(* IEC 61131-3 sources: generating_plc_code_with_llms/Code#1/Bard/first run, 20 files *)

(* ---- 14.st ---- *)
// 13.26s
// 2
FUNCTION FC1001(measuredValue: REAL, switchingValue: REAL, hysteresis: REAL): BOOL
VAR
previousOutput: BOOL; (* Flag indicating the previous output state )
switchingThreshold: REAL; ( Hysteresis-adjusted switching value *)

BEGIN
previousOutput := FALSE; (* Initialize previous output state to FALSE )
switchingThreshold := switchingValue * (1.0 - hysteresis / 100.0); ( Calculate the hysteresis-adjusted switching threshold *)

IF measuredValue >= switchingThreshold THEN
IF NOT previousOutput THEN
previousOutput := TRUE;
RETURN TRUE; (* Switch output on *)
END_IF;

RETURN previousOutput; (* Maintain output state *)
ELSE
IF previousOutput THEN
previousOutput := FALSE;
RETURN FALSE; (* Switch output off *)
END_IF;

RETURN previousOutput; (* Maintain output state *)
END_IF;
END_FUNCTION

(* ---- 15.st ---- *)
// 16.13s
// 1
FUNCTION FC1002(sensorInput: BOOL, manualSwitch: BOOL, hornOutput: BOOL, alarmOutput: BOOL, indicatorOutput: BOOL):
VAR
sensorState: BOOL; (* Flag indicating the current sensor state )
presenceTimer: TOF; ( Timer for object presence detection )
alarmEnabled: BOOL; ( Flag indicating whether the alarm is enabled *)

BEGIN
sensorState := sensorInput; (* Update sensor state *)

(* Update presence timer )
presenceTimer.IN := sensorState; ( Start/stop timer based on sensor state *)

(* Determine alarm state )
IF presenceTimer.Q AND presenceTimer.ET >= 3000 THEN
alarmEnabled := TRUE; ( Alarm condition met after 3 seconds )
ELSE
alarmEnabled := FALSE; ( Alarm condition not met or reset *)
END_IF;

(* Control outputs )
hornOutput := sensorState AND NOT alarmEnabled; ( Horn on for approach, off for alarm )
alarmOutput := alarmEnabled AND manualSwitch; ( Alarm on for alarm condition and manual switch on )
indicatorOutput := manualSwitch; ( Indicator on when manual switch is on *)
END_FUNCTION

VAR
  sensorInput: BOOL; (* Analog input value from ultrasonic sensor *)
  manualSwitch: BOOL; (* Input value from manual switch E_A *)
  hornOutput: BOOL; (* Output signal for horn P_HU *)
  alarmOutput: BOOL; (* Output signal for alarm P_AL *)
  indicatorOutput: BOOL; (* Output signal for indicator P1 *)

sensorInput := ReadAnalogInput(sensorInput);
manualSwitch := ReadInput(manualSwitchInput);

(* Call FC1002 to update outputs based on sensor input and manual switch *)
FC1002(sensorInput, manualSwitch, hornOutput, alarmOutput, indicatorOutput);

(* Control output devices based on updated output variables *)
WriteOutput(hornOutput, hornOutputDevice);
WriteOutput(alarmOutput, alarmOutputDevice);
WriteOutput(indicatorOutput, indicatorOutputDevice);

(* ---- 18.st ---- *)
// 7.53s
// 2
FUNCTION FC1003(inputValue: REAL; IN_MIN: REAL; IN_MAX: REAL; OUT_MIN: REAL; OUT_MAX: REAL): REAL
VAR
  rangeRatio: REAL; (* Ratio between input and output ranges *)
  scaledValue: REAL; (* Scaled input value *)

BEGIN
  (* Calculate range ratio *)
  rangeRatio := (OUT_MAX - OUT_MIN) / (IN_MAX - IN_MIN);

  (* Scale input value to output range *)
  scaledValue := (inputValue - IN_MIN) * rangeRatio;

  (* Adjust scaled value to output range limits *)
  IF scaledValue < OUT_MIN THEN
    scaledValue := OUT_MIN;
  ELSIF scaledValue > OUT_MAX THEN
    scaledValue := OUT_MAX;
  END_IF;

  (* Return scaled input value *)
  RETURN scaledValue;
END_FUNCTION

(* ---- 19.st ---- *)
// 9.82s
// 2
FUNCTION_BLOCK FB1005(
START: BOOL;
THICKNESS MD_1: BYTE;
V_MAX: REAL;
V_MIN: REAL;
D_MAX: BYTE;
D_MIN: BYTE;
)
VAR
currentThickness: REAL; (* Current thickness measurement )
largestThickness: REAL; ( Largest thickness measurement in current cycle )
smallestThickness: REAL; ( Smallest thickness measurement in current cycle )
rejectLight: BOOL; ( Flag indicating whether reject light is on *)

BEGIN
(* Initialize variables *)
largestThickness := 0.0;
smallestThickness := 0.0;
rejectLight := FALSE;

(* Continuously check for measurement start )
WHILE TRUE DO
IF START THEN
currentThickness := REAL(MD_1); ( Convert thickness value from flag double word *)

  (* Check for new largest or smallest thickness record *)
  IF currentThickness > largestThickness THEN
    largestThickness := currentThickness;
    D_MAX := MD_1; (* Update largest thickness output *)
  ELSIF currentThickness < smallestThickness THEN
    smallestThickness := currentThickness;
    D_MIN := MD_1;
  END_IF;

  (* Check for out-of-tolerance thickness *)
  IF currentThickness < V_MIN OR currentThickness > V_MAX THEN
    rejectLight := TRUE;

    (* Disable further measurement until restart *)
    START := FALSE;
  ELSE
    rejectLight := FALSE;
  END_IF;
END_IF;

(* Delay for 1 millisecond to avoid excessive processing *)
DELAY 0.001;
END_WHILE;
END_FUNCTION_BLOCK

VAR
  sensorS1: BOOL; (* Input signal from sensor S1 *)
  thicknessMD1: BYTE; (* Flag double word representing thickness measurement *)
  vMax: REAL; (* Maximum thickness tolerance *)
  vMin: REAL; (* Minimum thickness tolerance *)
  thicknessDMax: BYTE; (* Output flag double word for largest thickness *)
  thicknessDMin: BYTE; (* Output flag double word for smallest thickness *)

(* Call FB1005 to check plate thickness and update output variables *)
FB1005(sensorS1, thicknessMD1, vMax, vMin, thicknessDMax, thicknessDMin);

(* Update output devices based on output variables *)
WriteOutput(thicknessDMax, thicknessDMaxOutput);
WriteOutput(thicknessDMin, thicknessDMinOutput);

(* ---- 21.st ---- *)
// 14.54s
// 2
FUNCTION_BLOCK FB_BURNER(
  IN: BOOL;
  OVER_TEMP: BOOL;
  OIL_TEMP: BOOL;
  STAGE2: BOOL;
  RST: BOOL;
  PRE_HEAT_TIME: TIME;
  SAFETY_TIME: TIME;
  STAGE2_DELAY: TIME;
  MULTIPLE_IGNITION: BOOL;
  LOCKOUT_TIME: TIME;
  // Add other required parameters:
  PPR_IGNITION_TIME: TIME;
  PRE_VENTILATION_TIME: TIME;
  POST_IGNITION_TIME: TIME;
)
VAR
  // Internal states
  currentState: INT;
  lockOutTimer: TON;
  stage1Timer: TON;
  stage2Timer: TON;
  ignitionActive: BOOL;
  flameDetected: BOOL;
  error: INT;

BEGIN
  // Initialize variables
  lockOutTimer.IN := FALSE;
  stage1Timer.IN := FALSE;
  stage2Timer.IN := FALSE;
  ignitionActive := FALSE;
  flameDetected := FALSE;
  error := 0;

  // State machine transitions
  CASE currentState OF
    // Standby
    0: IF IN AND NOT OVER_TEMP THEN
        currentState := 1;
        PRE_HEAT := TRUE; // Start fuel oil warming
      END_IF;
    // Fuel oil warming
    1: IF OIL_TEMP THEN
        currentState := 2;
        ENGINE_ON := TRUE; // Start engine
        stage1Timer.IN := TRUE; // Start stage 1 timer
      ELSIF TIME_GT(TIME_DIFF(T_NOW(), START_TIME), PRE_HEAT_TIME) THEN
        error := 1;
        currentState := 10; // Go to error state
        FAIL := TRUE;
      END_IF;
    // Pre-ventilation
    2: IF TIME_GT(TIME_DIFF(T_NOW(), START_TIME), PRE_VENTILATION_TIME) THEN
        currentState := 3;
        IGNITION := TRUE; // Activate ignition
        ignitionActive := TRUE;
      ELSIF flameDetected THEN
        error := 3;
        currentState := 10; // Go to error state
        FAIL := TRUE;
      END_IF;
    // Ignition phase
    3: IF TIME_GT(TIME_DIFF(T_NOW(), START_TIME), PPR_IGNITION_TIME + SAFETY_TIME) THEN
        error := 4;
        currentState := 10; // Go to error state
        FAIL := TRUE;
      ELSIF flameDetected THEN
        currentState := 4;
        OIL_VALVE := TRUE; // Open oil valve
        ignitionActive := FALSE;
      END_IF;
    // Burning stage 1
    4: IF flameDetected THEN
        IF MULTIPLE_IGNITION AND NOT flameDetected THEN
          currentState := 3; // Restart ignition if flame breaks
        END_IF;
        IF STAGE2 AND TIME_GT(TIME_DIFF(T_NOW(), START_TIME), stage1Timer.PT + STAGE2_DELAY) THEN
          currentState := 5;
          stage2Timer.IN := TRUE; // Start stage 2 timer
        END_IF;
      ELSE
        error := 5;
        currentState := 10; // Go to error state
        FAIL := TRUE;
      END_IF;
    // Burning stage 2
    5: IF flameDetected THEN
        IF MULTIPLE_IGNITION AND NOT flameDetected THEN
          currentState := 3; // Restart ignition if flame breaks
        END_IF;
      ELSE
        error := 5;
        currentState := 10; // Go to error state
        FAIL := TRUE;
      END_IF;
    // Error state
    10: IF RST AND NOT OVER_TEMP THEN
        IF TIME_GT(TIME_DIFF(T_NOW(), START_TIME), LOCKOUT_TIME) THEN
          currentState := 0; // Reset and go to standby
        END_IF;
      ELSE
        lockOutTimer.IN := TRUE; // Start lockout timer
      END_IF;
  END_CASE;

  // Update outputs based on current state
  CASE currentState OF
    0: STATUS := 110;
    1: STATUS := 111;
    2: STATUS := 111;
    3: STATUS := 111;
    4: STATUS := 112;
    5: STATUS := 1

(* ---- 1.st ---- *)
//5.93s
//3
(* Program to manage two alarms *)

VAR
  xAlarm1: BOOL; (* Alarm 1 status *)
  xAlarm2: BOOL; (* Alarm 2 status *)
  xAllOn: BOOL; (* Set all alarms on *)
  xAllOff: BOOL; (* Set all alarms off *)

(* Main program *)
PROGRAM Main
BEGIN
  IF xAllOn THEN
    xAlarm1 := TRUE;
    xAlarm2 := TRUE;
  ELSIF xAllOff THEN
    xAlarm1 := FALSE;
    xAlarm2 := FALSE;
  END_IF;
END_PROGRAM

(* ---- 10.st ---- *)
//8.
// 2
(* Program to implement the sigmoid function *)

FUNCTION Sigmoid(x: REAL): REAL
BEGIN
  RETURN(1.0 / (1.0 + EXP(-x)));
END_FUNCTION

(* Main program *)
PROGRAM Main
VAR
  x: REAL; (* Input value *)
  y: REAL; (* Sigmoid function value *)

BEGIN
  x := 0.5; (* Example input value *)
  y := Sigmoid(x);
  WRITE('Sigmoid of', x, 'is', y);
END_PROGRAM

(* ---- 11.st ---- *)
//9.
// 2
(* Program to implement the sign function *)

FUNCTION Sign(x: REAL): REAL
BEGIN
  IF x > 0.0 THEN
    RETURN(1.0);
  ELSIF x < 0.0 THEN
    RETURN(-1.0);
  ELSE
    RETURN(0.0);
  END_IF;
END_FUNCTION

(* Main program *)
PROGRAM Main
VAR
  x: REAL; (* Input value *)
  signVal: REAL; (* Sign function value *)
BEGIN
  x := 5.0; (* Example input value *)
  signVal := Sign(x);
  WRITE('Sign of', x, 'is', signVal);

  x := -3.2;
  signVal := Sign(x);
  WRITE('Sign of', x, 'is', signVal);

  x := 0.0;
  signVal := Sign(x);
  WRITE('Sign of', x, 'is', signVal);
END_PROGRAM

(* ---- 12.st ---- *)
//8.59s
// 2
(* Program to implement the hyperbolic sine function using the exponential function *)

FUNCTION Sinh(x: REAL): REAL
BEGIN
  RETURN((EXP(x) - EXP(-x)) / 2.0);
END_FUNCTION

(* Main program *)
PROGRAM Main
VAR
  x: REAL; (* Input value *)
  sinhVal: REAL; (* Hyperbolic sine function value *)
BEGIN
  x := 1.0; (* Example input value *)
  sinhVal := Sinh(x);
  WRITE('Sinh of', x, 'is', sinhVal);
END_PROGRAM

(* ---- 13.st ---- *)
//9.83s
// 1
(* Program to search for the number 10 in a list of 100 random numbers )
VAR
randNum: INT; ( Random number )
numFound: BOOL; ( Flag indicating whether the number 10 has been found *)

(* Main program )
PROGRAM Main
BEGIN
numFound := FALSE; ( Initialize the flag *)

REPEAT
randNum := Random(101); (* Generate a random number between 0 and 100 (inclusive) *)
IF randNum = 10 THEN
  numFound := TRUE;
  EXIT; (* Exit the loop if the number 10 is found *)
END_IF;
UNTIL (numFound OR (i >= 100)); (* Continue searching until the number is found or the loop iterates 100 times *)

IF numFound THEN
WRITE('Number 10 found in the list');
ELSE
WRITE('Number 10 not found in the list');
END_IF;
END_PROGRAM

(* ---- 16.st ---- *)
//16.82s
// 2
(* Program to control a simple traffic light with two lights *)

VAR
  cycleTimer: TON; (* Timer for the traffic light cycle *)
  northGreen: BOOL; (* Flag indicating North light is green *)
  northYellow: BOOL; (* Flag indicating North light is yellow *)
  northRed: BOOL; (* Flag indicating North light is red *)
  eastGreen: BOOL; (* Flag indicating East light is green *)
  eastYellow: BOOL; (* Flag indicating East light is yellow *)
  eastRed: BOOL; (* Flag indicating East light is red *)

(* Main program *)
PROGRAM Main
BEGIN
  (* Initialize timer and output variables *)
  cycleTimer.IN := TRUE; (* Start the timer *)
  northGreen := FALSE;
  northYellow := FALSE;
  northRed := TRUE;
  eastGreen := FALSE;
  eastYellow := FALSE;
  eastRed := TRUE;

  REPEAT
    (* Update output variables based on timer state and elapsed time *)
    IF cycleTimer.Q THEN
      IF cycleTimer.ET >= 0 AND cycleTimer.ET < 5000 THEN
        northGreen := TRUE;
        northYellow := FALSE;
        northRed := FALSE;
        eastGreen := FALSE;
        eastYellow := FALSE;
        eastRed := TRUE;
      ELSIF cycleTimer.ET >= 5000 AND cycleTimer.ET < 5500 THEN
        northGreen := FALSE;
        northYellow := TRUE;
        northRed := FALSE;
        eastGreen := FALSE;
        eastYellow := FALSE;
        eastRed := TRUE;
      ELSIF cycleTimer.ET >= 5500 AND cycleTimer.ET < 9500 THEN
        northGreen := FALSE;
        northYellow := FALSE;
        northRed := TRUE;
        eastGreen := TRUE;
        eastYellow := FALSE;
        eastRed := FALSE;
      ELSIF cycleTimer.ET >= 9500 AND cycleTimer.ET < 10000 THEN
        northGreen := FALSE;
        northYellow := FALSE;
        northRed := TRUE;
        eastGreen := FALSE;
        eastYellow := TRUE;
        eastRed := FALSE;
      ELSE
        (* Reset timer and output variables for next cycle *)
        cycleTimer.IN := TRUE;
        northGreen := FALSE;
        northYellow := FALSE;
        northRed := TRUE;
        eastGreen := FALSE;
        eastYellow := FALSE;
        eastRed := TRUE;
      END_IF;
    END_IF;
  UNTIL FALSE; (* Loop indefinitely *)
END_PROGRAM

(* ---- 2.st ---- *)
//8.86s
//2
(* Program to calculate the binomial coefficient *)

VAR
  n: INT; (* Number of items *)
  k: INT; (* Number of choices *)
  result: INT; (* Binomial coefficient *)

(* Main program *)
PROGRAM Main
BEGIN
  n := 10;
  k := 2;
  result := BinomialCoefficient(n, k);
  WRITE('The binomial coefficient of', n, 'choose', k, 'is', result);
END_PROGRAM

(* Function to calculate the binomial coefficient *)
FUNCTION BinomialCoefficient(n: INT; k: INT): INT
VAR
  i: INT;
  temp: INT;
BEGIN
  IF k > n THEN
    RETURN(0);
  END_IF;
  IF k = 0 OR k = n THEN
    RETURN(1);
  END_IF;
  temp := 1;
  FOR i := 1 TO k DO
    temp := temp * (n - i + 1);
    temp := temp / i;
  END_FOR;
  RETURN(temp);
END_FUNCTION

(* ---- 20.st ---- *)
// 10.12s
// 2
VAR
  lastI1Value: BOOL; (* Boolean variable to store the previous value of I1 *)
  lastI2Value: BOOL; (* Boolean variable to store the previous value of I2 *)
  interlockTime: TIMER; (* Timer for interlock dead time *)
  outputQ1: BOOL; (* Boolean variable to control output Q1 *)
  outputQ2: BOOL; (* Boolean variable to control output Q2 *)

BEGIN
  interlockTime := TIMER;
  lastI1Value := FALSE;
  lastI2Value := FALSE;

  WHILE TRUE DO
    IF I1 THEN
      (* Check if interlock time is over *)
      IF (interlockTime.ET >= TL) THEN
        outputQ1 := TRUE;
      END_IF;
    ELSE
      outputQ1 := FALSE;
    END_IF;

    IF I2 THEN
      (* Check if interlock time is over *)
      IF (interlockTime.ET >= TL) THEN
        outputQ2 := TRUE;
      END_IF;
    ELSE
      outputQ2 := FALSE;
    END_IF;

    (* Update interlock time *)
    interlockTime.IN := FALSE;

    (* Delay for 1 millisecond to avoid excessive processing *)
    DELAY 0.001;
  END_WHILE;

  (* Update output devices based on output variables *)
  WriteOutput(outputQ1, outputQ1Output);
  WriteOutput(outputQ2, outputQ2Output);

(* ---- 3.st ---- *)
//8.29s
//2
(* Program to calculate a Fibonacci number *)

VAR
  n: INT; (* Fibonacci number to calculate *)
  result: INT; (* Calculated Fibonacci number *)

(* Main program *)
PROGRAM Main
BEGIN
  n := 10;
  result := Fibonacci(n);
  WRITE('The Fibonacci number of', n, 'is', result);
END_PROGRAM

(* Function to calculate a Fibonacci number *)
FUNCTION Fibonacci(n: INT): INT
BEGIN
  IF n = 0 THEN
    RETURN(0);
  ELSIF n = 1 THEN
    RETURN(1);
  ELSE
    RETURN(Fibonacci(n - 1) + Fibonacci(n - 2));
  END_IF;
END_FUNCTION

(* ---- 4.st ---- *)
//12.27s
// 2
(* Program to monitor fill level in a container *)

VAR
  fillLevelAnalog: INT; (* Analog value of fill level (0-32767) *)
  fillLevelPercent: REAL; (* Fill level in percent (0-100%) *)
  isLow: BOOL; (* Fill level is low *)
  isOk: BOOL; (* Fill level is ok *)
  isHigh: BOOL; (* Fill level is high *)
  isWarningHornOn: BOOL; (* Warning horn is on *)

(* Main program *)
PROGRAM Main
BEGIN
  fillLevelAnalog := ReadAnalogInput();
  fillLevelPercent := ConvertAnalogToPercent(fillLevelAnalog);

  CASE fillLevelPercent OF
    0.0 TO 1.0:
      isLow := TRUE;
      isOk := FALSE;
      isHigh := FALSE;
      isWarningHornOn := TRUE;
    1.1 TO 30.0:
      isLow := FALSE;
      isOk := TRUE;
      isHigh := FALSE;
      isWarningHornOn := FALSE;
    30.1 TO 90.0:
      isLow := FALSE;
      isOk := TRUE;
      isHigh := FALSE;
      isWarningHornOn := FALSE;
    90.1 TO 100.0:
      isLow := FALSE;
      isOk := FALSE;
      isHigh := TRUE;
      isWarningHornOn := FALSE;
  END_CASE;

  WriteOutput(isLow, isOk, isHigh, isWarningHornOn);
END_PROGRAM

(* Function to convert analog value to percent *)
FUNCTION ConvertAnalogToPercent(analogValue: INT): REAL
VAR
  percent: REAL;
BEGIN
  percent := (REAL)analogValue / 32767.0 * 100.0;
  RETURN(percent);
END_FUNCTION

(* ---- 5.st ---- *)
//12.0s
// 2
(* Program to control a gate *)

VAR
  Start_Loop: BOOL; (* Start loop flag *)
  One_Hour_Timer: TIME; (* One-hour timer *)
  Gate_Open: BOOL; (* Gate open flag *)
  Auth_String: STRING(50); (* Authentication string *)
  My_Defined_Str: STRING(50) := 'my_defined_str'; (* My defined authentication string *)
  App_Or_Car_Sensed: BOOL; (* App or car sensed flag *)

(* Main program *)
PROGRAM Main
BEGIN
  IF NOT Start_Loop THEN
    TON(PT:= 1h, IN:= TRUE, OUT:= One_Hour_Timer.Q); (* Start one-hour timer *)
  END_IF;

  IF One_Hour_Timer.Q AND Gate_Open THEN
    Gate_Open := FALSE; (* Close gate if timer timed out and gate is still open *)
  END_IF;

  IF App_Or_Car_Sensed THEN
    CASE Auth_String OF
      My_Defined_Str: Gate_Open := TRUE; (* Open gate if authentication string matches *)
      ELSE: Gate_Open := FALSE; (* Keep gate closed if authentication string does not match *)
    END_CASE;
  END_IF;

  WriteOutput(Gate_Open); (* Write gate open flag to output *)
END_PROGRAM

(* ---- 6.st ---- *)
//23.35s
// 2 nicht alle Variablen deklariert
(* Program to control a crane lift *)

VAR
  diConvTop: BOOL; (* Light barrier top conveyor belt *)
  diConvBottom: BOOL; (* Light barrier bottom conveyor belt *)
  doConvTop: BOOL; (* Conveyor belt top *)
  doConvBottom: BOOL; (* Conveyor belt bottom *)
  doLiftTop: BOOL; (* Lift top *)
  doLiftBottom: BOOL; (* Lift bottom *)
  doConvLift: BOOL; (* Lift conveyor belt *)
  diLiftTop: BOOL; (* Lift position top *)
  diLiftBottom: BOOL; (* Lift position bottom *)
  diLiftUnload: BOOL; (* Lift position unload *)
  liftRequested: BOOL; (* Lift requested flag *)

(* Main program *)
PROGRAM Main
BEGIN
  IF diConvTop THEN
    doConvTop := FALSE; (* Stop top conveyor belt when light barrier is activated *)
    IF NOT liftRequested THEN
      doLiftTop := TRUE; (* Move lift to top position if not already requested *)
      liftRequested := TRUE; (* Mark lift as requested *)
    END_IF;
  END_IF;

  IF diConvBottom THEN
    doConvBottom := FALSE; (* Stop bottom conveyor belt when light barrier is activated *)
    IF NOT liftRequested THEN
      doLiftBottom := TRUE; (* Move lift to bottom position if not already requested *)
      liftRequested := TRUE; (* Mark lift as requested *)
    END_IF;
  END_IF;

  IF diLiftTop AND liftRequested THEN
    doConvLift := TRUE; (* Start lift conveyor belt when lift is in position and requested *)
  END_IF;

  IF diBoxLift THEN
    doConvLift := FALSE; (* Stop lift conveyor belt when box reaches lift *)
  END_IF;

  IF diLiftUnload THEN
    doLiftUnload := TRUE; (* Move lift to unload position when it reaches the position *)
  END_IF;

  IF diLiftUnload AND NOT diBoxLift THEN
    liftRequested := FALSE; (* Reset lift requested flag when box leaves lift *)
  END_IF;
END_PROGRAM

(* ---- 7.st ---- *)
//12.5s
// 2
(* Program to calculate total load and average load *)

CONST
  NUM_LOAD_RECEPTORS = 5; (* Number of load receptors *)
  MAX_ANALOG_VALUE = 32767; (* Maximum analog input value *)

VAR
  loadValues: ARRAY[0..NUM_LOAD_RECEPTORS - 1] OF REAL; (* Array to store load values *)
  totalLoad: REAL; (* Total load *)
  averageLoad: REAL; (* Average load *)

(* Main program *)
PROGRAM Main
BEGIN
  (* Read load values from analog inputs *)
  FOR i := 0 TO NUM_LOAD_RECEPTORS - 1 DO
    loadValues[i] := ReadAnalogInput(i) / MAX_ANALOG_VALUE;
  END_FOR;

  (* Calculate total load *)
  totalLoad := 0.0;
  FOR i := 0 TO NUM_LOAD_RECEPTORS - 1 DO
    totalLoad := totalLoad + loadValues[i];
  END_FOR;

  (* Calculate average load *)
  averageLoad := totalLoad / NUM_LOAD_RECEPTORS;

  (* Write total load and average load to outputs *)
  WriteOutput(totalLoad, averageLoad);
END_PROGRAM

(* ---- 8.st ---- *)
//11.18s
// 2
(* Program to implement the Lambert W function *)

CONST
  EPSILON = 1e-6; (* Tolerance for the iteration *)
  MAX_ITERATIONS = 100; (* Maximum number of iterations *)

(* Function to calculate the Lambert W function *)
FUNCTION LambertW(x: REAL): REAL
VAR
  y: REAL; (* Initial approximation *)
  w: REAL; (* Lambert W function value *)
  i: INT; (* Iteration counter *)

BEGIN
  y := log(x);
  FOR i := 1 TO MAX_ITERATIONS DO
    w := y - x * EXP(-y);
    IF ABS(w - y) < EPSILON THEN
      RETURN(w);
    END_IF;
    y := w;
  END_FOR;
  RETURN(0.0); (* No convergence *)
END_FUNCTION

(* Main program *)
PROGRAM Main
VAR
  x: REAL; (* Input value *)
  w: REAL; (* Lambert W function value *)

BEGIN
  x := 1.5; (* Example input value *)
  w := LambertW(x);
  WRITE('Lambert W of', x, 'is', w);
END_PROGRAM

(* ---- 9.st ---- *)
//9.16s
// 2
(* Program to check whether a year is a leap year *)

VAR
  YEAR: INT; (* Year to check *)
  isLeapYear: BOOL; (* Flag indicating whether the year is a leap year *)

(* Main program *)
PROGRAM Main
BEGIN
  YEAR := 2020; (* Example year *)
  isLeapYear := ((YEAR MOD 4 = 0) AND (YEAR MOD 100 <> 0)) OR (YEAR MOD 400 = 0);
  IF isLeapYear THEN
    WRITE(YEAR, 'is a leap year');
  ELSE
    WRITE(YEAR, 'is not a leap year');
  END_IF;
END_PROGRAM
